(* PLC project Generated.project, CODESYS CODESYS V3.5 SP19 Patch 1 *)
(* stored: creationDateTime 2026-09-06T13:00:42.512422, modificationDateTime 2026-09-06T13:00:42.512422 *)

(* values of E_ProgramSequence: NONE: Aucune séquence active; MAIN_CYCLE: Cycle semi-automatique principal (FB_Cycle); DIVE_SEARCH: Recherche de fond Kobold (réservé future migration); EXTRACTION: Séquence d'extraction (réservé future migration) *)

{attribute 'qualified_only'}
{attribute 'strict'}
TYPE E_ProgramSequence : (NONE := 0, MAIN_CYCLE := 1, DIVE_SEARCH := 2, EXTRACTION := 3);
END_TYPE
